TYPE E_RecvStates :
(**************************************************************************************
 * 	AUTHOR		Swisslog
 * 	LIBRARY		Data types/02_Library/02_Communication/TCP-Driver
 *	RELEASE		1.0.0
 * ------------------------------------------------------------------------------------
 * 	Revision History: 
 *
 * 	VERSION		DATE		INITIALS	DESCRIPTION
 *	0.1		07.09.2011	swl		initial version
 **************************************************************************************)
(
	RECV_IDLE,
	RECV_WAIT,
	RECV_ERROR
);
END_TYPE

(* stored: Version 1.1.0.1, ProductVersion 3.1.4020.6
   DUT E_RecvStates: Id {91cc4fc0-d4d6-49f7-ac9f-7fb652024a41} *)
